PROGRAM PRG_Test
VAR
	FC_AddTests : FC_Add_Test;
	
	
END_VAR

TCUnit.RUN();

END_PROGRAM

(* stored: Version 1.1.0.1
   POU PRG_Test: Id {2ff844ec-0d5f-42bf-a856-8e8ada83d934}, SpecialFunc None *)
